{attribute 'qualified_only'}
VAR_GLOBAL CONSTANT
    rMinWeightConstant      : REAL  := 10.0;
    rMaxWeightConstant  : REAL  := 550.0;
END_VAR

(* stored: Version 1.1.0.1, ProductVersion 3.1.4024.16
   GVL WeightRange: Id {7ebdb4ac-820c-4f81-86ea-e66de6307b8b} *)
